FUNCTION_BLOCK N_TBL (* Gets the Nth element from a list of strings *)
  (* Standard: 61499-1; Classification: Math *)
  (* Version 0.1, 2008-06-04, JHC, Holobloc Inc, Updated DOCTYPE. *)
  (* Version 0.0, 2000-04-21, JHC, Rockwell Automation *)
  (* Compiler header: package fb.rt.math; *)
  (* Compiler Java IBM VisualAge 3.0 *)
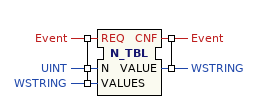
  EVENT_INPUT
    REQ WITH N, VALUES; (* Table Lookup *)
  END_EVENT
  EVENT_OUTPUT
    CNF WITH VALUE; (* Lookup Result *)
  END_EVENT
  VAR_INPUT
    N : UINT; (* Key for Lookup *)
    VALUES : WSTRING; (* Comma-separated List of Values *)
  END_VAR
  VAR_OUTPUT
    VALUE : WSTRING; (* Lookup Result,Empty if Lookup Failed *)
  END_VAR
  SERVICE APPLICATION/N_TBL
    SEQUENCE normal_lookup
      APPLICATION.REQ(KEY) -> APPLICATION.CNF(VALUE);
    END_SEQUENCE
    SEQUENCE lookup_error
      APPLICATION.REQ(SD) -> APPLICATION.CNF("");
    END_SEQUENCE
  END_SERVICE
END_FUNCTION_BLOCK
